FUNCTION ArrayContains : BOOL
VAR_IN_OUT
	arr : ARRAY[*] OF INT;
END_VAR
VAR_INPUT
	value : INT;
END_VAR
VAR
	i : DINT;
END_VAR

FOR i:=0 TO UPPER_BOUND(arr, 1) BY 1 DO
	IF arr[i] = value THEN
		ArrayContains := TRUE;
		RETURN;
	END_IF
END_FOR

ArrayContains := FALSE;

END_FUNCTION

(* stored: Version 1.1.0.1, ProductVersion 3.1.4024.11
   POU ArrayContains: Id {0aa87cf0-ef8b-408f-ace1-ccf703741a9c}, SpecialFunc None *)
